{attribute 'qualified_only'}
VAR_GLOBAL
	B1 :BOOL; // Endschalter Offen
	B2: BOOL;     // Endschalter Geschlossen
	B3: BOOL;     // Lichtschranke
	S1: BOOL;     // Taster "Halt"
	S2: BOOL;     // Taster "Öffnen"
	S3: BOOL;      // Taster "Schliessen"
END_VAR

(* stored: Version 1.1.0.1, ProductVersion 3.1.4024.5
   GVL SimDI: Id {c2d05302-d374-4f85-80dd-41006a3e3277} *)
